Universal Robots PolyScope program: ur_comm_test.urp

Program ur_comm_test (installation=default directory=/home/ur/ursim-current/programs createdIn=5.5.1.82186 lastSavedIn=5.9.4.1031232 robotSerialNumber=20195599999)
Calibrated DH parameters: a=[0, -0.425, -0.3922, 0, 0, 0]; d=[0.1625, 0, 0, 0.1333, 0.0997, 0.0996]; alpha=[1.570796, 0, 0, 1.570796, -1.570796, 0]; deltaTheta=[0, 0, 0, 0, 0, 0]
InitVariablesNode variables(variable(name=Counter, expression=0))
Robot Program (runOnlyOnce=false)
  MoveJ speed 15 deg/s, acceleration 15 deg/s^2 (useActiveTCP=true) feature=Base
    Waypoint robot_pose_1: TCP in base x=537.26 y=181.734 z=515.774 mm, rx=-3.103 ry=-0.0398 rz=-0.0836 rad; joints [32.056, -97.252, -79.274, -89.771, 90.491, -59.17] deg; TCP offset x=0 y=0 z=0 mm, rx=0 ry=0 rz=0 rad
  Script: write_output_integer_register(24,0)
  Script: write_output_boolean_register(64,False)
  Wait Condition expression=read_input_boolean_register(65)
  Script: read_input_boolean_register(65)
  'Reading x,y,z,rx,ry,rz valuse'
  x := read_input_float_register(24)
  y := read_input_float_register(25)
  z := read_input_float_register(26)
  rx := read_input_float_register(27)
  ry := read_input_float_register(28)
  rz := read_input_float_register(29)
  start_pose := get_actual_tcp_pose()
  target_pose := p[x,y,z,rx,ry,rz]
  Script: movel(target_pose, a=1.0, v=1.0, t=0, r=0)
  Wait Condition expression=pose_dist(target_pose, get_actual_tcp_pose())<0.01
  Wait Sleep waitTime=0.5
  Script: write_output_integer_register(24,-1)
  MoveJ speed 15 deg/s, acceleration 15 deg/s^2 (useActiveTCP=true) feature=Base
    Waypoint robot_pose_1: TCP in base x=537.26 y=181.734 z=515.774 mm, rx=-3.103 ry=-0.0398 rz=-0.0836 rad; joints [32.056, -97.252, -79.274, -89.771, 90.491, -59.17] deg
  Halt
SuppressedNode
  SubProgram capture_hand_eye (keepSynchronizedWithDisk=false)
    Wait Sleep waitTime=2
    Counter := Counter+1
    SuppressedNode
      Set ExpressionOutput pin=GP_int_out[24]; expression=Counter
    Script: write_output_integer_register(24,Counter)
    SuppressedNode
      Set DigitalOutput pin=GP_bool_out[64]; digitalValue=1
    Script: write_output_boolean_register(64, True)
    Wait Condition expression=read_input_boolean_register(64)
    SuppressedNode
      Set DigitalOutput pin=GP_bool_out[64]; digitalValue=0
    Script: write_output_boolean_register(64, False)
